(* IEC 61131-3 sources: AXOpen/src/components.rexroth.tightening/ctrl/src/TemplateComponent (part 2) *)

                    IF TRUE THEN
                        THIS.CallTimers(FALSE);
                        _progress := 346;
                    END_IF;
                END_IF;

                IF _progress = 346 THEN                                                                                     // TemplateTask_10steps_5 running: , <add the detailed description of the current action 7>
                    TaskMessenger.ActivateOnCondition(ULINT#546, _infoTimer.output, eAxoMessageCategory#Warning);
                    IF _infoTimer.output THEN
                        Status.Error.Id := UINT#546;
                    END_IF;

                    IF TRUE THEN
                        THIS.CallTimers(FALSE);
                        _progress := 347;
                    END_IF;
                END_IF;

                IF _progress = 347 THEN                                                                                     // TemplateTask_10steps_5 running: , <add the detailed description of the current action 8>
                    TaskMessenger.ActivateOnCondition(ULINT#547, _infoTimer.output, eAxoMessageCategory#Warning);
                    IF _infoTimer.output THEN
                        Status.Error.Id := UINT#547;
                    END_IF;

                    IF TRUE THEN
                        THIS.CallTimers(FALSE);
                        _progress := 348;
                    END_IF;
                END_IF;

                IF _progress = 348 THEN                                                                                     // TemplateTask_10steps_5 running: , <add the detailed description of the current action 9>
                    TaskMessenger.ActivateOnCondition(ULINT#548, _infoTimer.output, eAxoMessageCategory#Warning);
                    IF _infoTimer.output THEN
                        Status.Error.Id := UINT#548;
                    END_IF;

                    IF TRUE THEN
                        THIS.CallTimers(FALSE);
                        _progress := 349;
                    END_IF;
                END_IF;

                IF _progress = 349 THEN                                                                                     // TemplateTask_10steps_5 running: , <add the detailed description of the current action 10>
                    TemplateTask_10steps_5.DoneWhen(TRUE);
                END_IF;

                THIS.CallTimers(TRUE);

                TemplateTask_10steps_5.ThrowWhen(_errorTimer.output);
                Status.Action.Id := TO_UINT(_progress);
                TemplateTask_10steps_5.ThrowWhen(TemplateTask_10steps_5.Duration >= Config.ErrorTime ,'TemplateTask_10steps_5 error.');
            END_IF;
            IF TemplateTask_10steps_5.DoneReached() THEN
                Status.Action.Id :=  UINT#141;
                Status.Error.Id :=  UINT#0;
            ELSIF TemplateTask_10steps_5.ErrorOccured() THEN
                Status.Action.Id :=  UINT#940;
                Status.Error.Id  :=  UINT#940;
            ELSIF TemplateTask_10steps_5.AbortTriggered()THEN
                Status.Action.Id :=  UINT#941;
                Status.Error.Id  :=  UINT#941;
            END_IF;
            Messenger.ActivateOnCondition(ULINT#940,TemplateTask_10steps_5.HasError(), eAxoMessageCategory#Error);
            Messenger.ActivateOnCondition(ULINT#941,TemplateTask_10steps_5.IsAborted(), eAxoMessageCategory#Error);
            Messenger.ActivateOnCondition(ULINT#142,TemplateTask_10steps_5.RestoreTriggered() , eAxoMessageCategory#Error);
            IF TemplateTask_10steps_5.RestoreTriggered() AND _progress >= 340 AND _progress <= 349  THEN
                Status.Action.Id :=  UINT#142;
                _progress := 0;
            END_IF;
            //**************************************************

            //*************TemplateTask_10steps_6***************
            TemplateTask_10steps_6.SetIsDisabled(FALSE);
            IF TemplateTask_10steps_6.StartTriggered() THEN
                Status.Action.Id :=  UINT#150;
            END_IF;
            Messenger.ActivateOnCondition(ULINT#150,TemplateTask_10steps_6.IsBusy(), eAxoMessageCategory#Info);
            Messenger.ActivateOnCondition(ULINT#151,TemplateTask_10steps_6.IsDone(), eAxoMessageCategory#Info);
            IF TemplateTask_10steps_6.Execute(THIS) THEN
                IF _progress = 0 THEN
                    Status.Error.Id := UINT#0;
                    TaskMessenger.Restore();
                    THIS.CallTimers(FALSE);
                    _progress := 350;
                END_IF;

                IF _progress = 350 THEN                                                                                     // TemplateTask_10steps_6 running: , <add the detailed description of the current action 1>
                    TaskMessenger.ActivateOnCondition(ULINT#550, _infoTimer.output, eAxoMessageCategory#Warning);
                    IF _infoTimer.output THEN
                        Status.Error.Id := UINT#550;
                    END_IF;

                    IF TRUE THEN
                        THIS.CallTimers(FALSE);
                        _progress := 351;
                    END_IF;
                END_IF;

                IF _progress = 351 THEN                                                                                     // TemplateTask_10steps_6 running: , <add the detailed description of the current action 2>
                    TaskMessenger.ActivateOnCondition(ULINT#551, _infoTimer.output, eAxoMessageCategory#Warning);
                    IF _infoTimer.output THEN
                        Status.Error.Id := UINT#551;
                    END_IF;

                    IF TRUE THEN
                        THIS.CallTimers(FALSE);
                        _progress := 352;
                    END_IF;
                END_IF;

                IF _progress = 352 THEN                                                                                     // TemplateTask_10steps_6 running: , <add the detailed description of the current action 3>
                    TaskMessenger.ActivateOnCondition(ULINT#552, _infoTimer.output, eAxoMessageCategory#Warning);
                    IF _infoTimer.output THEN
                        Status.Error.Id := UINT#552;
                    END_IF;

                    IF TRUE THEN
                        THIS.CallTimers(FALSE);
                        _progress := 335;
                    END_IF;
                END_IF;

                IF _progress = 353 THEN                                                                                     // TemplateTask_10steps_6 running: , <add the detailed description of the current action 4>
                    TaskMessenger.ActivateOnCondition(ULINT#553, _infoTimer.output, eAxoMessageCategory#Warning);
                    IF _infoTimer.output THEN
                        Status.Error.Id := UINT#553;
                    END_IF;

                    IF TRUE THEN
                        THIS.CallTimers(FALSE);
                        _progress := 354;
                    END_IF;
                END_IF;

                IF _progress = 354 THEN                                                                                     // TemplateTask_10steps_6 running: , <add the detailed description of the current action 5>
                    TaskMessenger.ActivateOnCondition(ULINT#554, _infoTimer.output, eAxoMessageCategory#Warning);
                    IF _infoTimer.output THEN
                        Status.Error.Id := UINT#554;
                    END_IF;

                    IF TRUE THEN
                        THIS.CallTimers(FALSE);
                        _progress := 355;
                    END_IF;
                END_IF;

                IF _progress = 355 THEN                                                                                     // TemplateTask_10steps_6 running: , <add the detailed description of the current action 6>
                    TaskMessenger.ActivateOnCondition(ULINT#555, _infoTimer.output, eAxoMessageCategory#Warning);
                    IF _infoTimer.output THEN
                        Status.Error.Id := UINT#555;
                    END_IF;

                    IF TRUE THEN
                        THIS.CallTimers(FALSE);
                        _progress := 356;
                    END_IF;
                END_IF;

                IF _progress = 356 THEN                                                                                     // TemplateTask_10steps_6 running: , <add the detailed description of the current action 7>
                    TaskMessenger.ActivateOnCondition(ULINT#556, _infoTimer.output, eAxoMessageCategory#Warning);
                    IF _infoTimer.output THEN
                        Status.Error.Id := UINT#556;
                    END_IF;

                    IF TRUE THEN
                        THIS.CallTimers(FALSE);
                        _progress := 357;
                    END_IF;
                END_IF;

                IF _progress = 357 THEN                                                                                     // TemplateTask_10steps_6 running: , <add the detailed description of the current action 8>
                    TaskMessenger.ActivateOnCondition(ULINT#557, _infoTimer.output, eAxoMessageCategory#Warning);
                    IF _infoTimer.output THEN
                        Status.Error.Id := UINT#557;
                    END_IF;

                    IF TRUE THEN
                        THIS.CallTimers(FALSE);
                        _progress := 358;
                    END_IF;
                END_IF;

                IF _progress = 358 THEN                                                                                     // TemplateTask_10steps_6 running: , <add the detailed description of the current action 9>
                    TaskMessenger.ActivateOnCondition(ULINT#558, _infoTimer.output, eAxoMessageCategory#Warning);
                    IF _infoTimer.output THEN
                        Status.Error.Id := UINT#558;
                    END_IF;

                    IF TRUE THEN
                        THIS.CallTimers(FALSE);
                        _progress := 359;
                    END_IF;
                END_IF;

                IF _progress = 359 THEN                                                                                     // TemplateTask_10steps_6 running: , <add the detailed description of the current action 10>
                    TemplateTask_10steps_6.DoneWhen(TRUE);
                END_IF;

                THIS.CallTimers(TRUE);

                TemplateTask_10steps_6.ThrowWhen(_errorTimer.output);
                Status.Action.Id := TO_UINT(_progress);
                TemplateTask_10steps_6.ThrowWhen(TemplateTask_10steps_6.Duration >= Config.ErrorTime ,'TemplateTask_10steps_6 error.');
            END_IF;
            IF TemplateTask_10steps_6.DoneReached() THEN
                Status.Action.Id :=  UINT#151;
                Status.Error.Id :=  UINT#0;
            ELSIF TemplateTask_10steps_6.ErrorOccured() THEN
                Status.Action.Id :=  UINT#950;
                Status.Error.Id  :=  UINT#950;
            ELSIF TemplateTask_10steps_6.AbortTriggered()THEN
                Status.Action.Id :=  UINT#951;
                Status.Error.Id  :=  UINT#951;
            END_IF;
            Messenger.ActivateOnCondition(ULINT#950,TemplateTask_10steps_6.HasError(), eAxoMessageCategory#Error);
            Messenger.ActivateOnCondition(ULINT#951,TemplateTask_10steps_6.IsAborted(), eAxoMessageCategory#Error);
            Messenger.ActivateOnCondition(ULINT#152,TemplateTask_10steps_6.RestoreTriggered() , eAxoMessageCategory#Error);
            IF TemplateTask_10steps_6.RestoreTriggered() AND _progress >= 350 AND _progress <= 359  THEN
                Status.Action.Id :=  UINT#152;
                _progress := 0;
            END_IF;
            //**************************************************

            //*************TemplateTask_20steps_1***************
            TemplateTask_20steps_1.SetIsDisabled(FALSE);
            IF TemplateTask_20steps_1.StartTriggered() THEN
                Status.Action.Id :=  UINT#160;
            END_IF;
            Messenger.ActivateOnCondition(ULINT#160,TemplateTask_20steps_1.IsBusy(), eAxoMessageCategory#Info);
            Messenger.ActivateOnCondition(ULINT#161,TemplateTask_20steps_1.IsDone(), eAxoMessageCategory#Info);
            IF TemplateTask_20steps_1.Execute(THIS) THEN
                IF _progress = 0 THEN
                    Status.Error.Id := UINT#0;
                    TaskMessenger.Restore();
                    THIS.CallTimers(FALSE);
                    _progress := 360;
                END_IF;

                IF _progress = 360 THEN                                                                                     // TemplateTask_20steps_1 running: , <add the detailed description of the current action 1>
                    TaskMessenger.ActivateOnCondition(ULINT#560, _infoTimer.output, eAxoMessageCategory#Warning);
                    IF _infoTimer.output THEN
                        Status.Error.Id := UINT#560;
                    END_IF;

                    IF TRUE THEN
                        THIS.CallTimers(FALSE);
                        _progress := 361;
                    END_IF;
                END_IF;

                IF _progress = 361 THEN                                                                                     // TemplateTask_20steps_1 running: , <add the detailed description of the current action 2>
                    TaskMessenger.ActivateOnCondition(ULINT#561, _infoTimer.output, eAxoMessageCategory#Warning);
                    IF _infoTimer.output THEN
                        Status.Error.Id := UINT#561;
                    END_IF;

                    IF TRUE THEN
                        THIS.CallTimers(FALSE);
                        _progress := 362;
                    END_IF;
                END_IF;

                IF _progress = 362 THEN                                                                                     // TemplateTask_20steps_1 running: , <add the detailed description of the current action 3>
                    TaskMessenger.ActivateOnCondition(ULINT#562, _infoTimer.output, eAxoMessageCategory#Warning);
                    IF _infoTimer.output THEN
                        Status.Error.Id := UINT#562;
                    END_IF;

                    IF TRUE THEN
                        THIS.CallTimers(FALSE);
                        _progress := 363;
                    END_IF;
                END_IF;

                IF _progress = 363 THEN                                                                                     // TemplateTask_20steps_1 running: , <add the detailed description of the current action 4>
                    TaskMessenger.ActivateOnCondition(ULINT#563, _infoTimer.output, eAxoMessageCategory#Warning);
                    IF _infoTimer.output THEN
                        Status.Error.Id := UINT#563;
                    END_IF;

                    IF TRUE THEN
                        THIS.CallTimers(FALSE);
                        _progress := 364;
                    END_IF;
                END_IF;

                IF _progress = 364 THEN                                                                                     // TemplateTask_20steps_1 running: , <add the detailed description of the current action 5>
                    TaskMessenger.ActivateOnCondition(ULINT#564, _infoTimer.output, eAxoMessageCategory#Warning);
                    IF _infoTimer.output THEN
                        Status.Error.Id := UINT#564;
                    END_IF;

                    IF TRUE THEN
                        THIS.CallTimers(FALSE);
                        _progress := 365;
                    END_IF;
                END_IF;

                IF _progress = 365 THEN                                                                                     // TemplateTask_20steps_1 running: , <add the detailed description of the current action 6>
                    TaskMessenger.ActivateOnCondition(ULINT#565, _infoTimer.output, eAxoMessageCategory#Warning);
                    IF _infoTimer.output THEN
                        Status.Error.Id := UINT#565;
                    END_IF;

                    IF TRUE THEN
                        THIS.CallTimers(FALSE);
                        _progress := 366;
                    END_IF;
                END_IF;

                IF _progress = 366 THEN                                                                                     // TemplateTask_20steps_1 running: , <add the detailed description of the current action 7>
                    TaskMessenger.ActivateOnCondition(ULINT#566, _infoTimer.output, eAxoMessageCategory#Warning);
                    IF _infoTimer.output THEN
                        Status.Error.Id := UINT#566;
                    END_IF;

                    IF TRUE THEN
                        THIS.CallTimers(FALSE);
                        _progress := 367;
                    END_IF;
                END_IF;

                IF _progress = 367 THEN                                                                                     // TemplateTask_20steps_1 running: , <add the detailed description of the current action 8>
                    TaskMessenger.ActivateOnCondition(ULINT#567, _infoTimer.output, eAxoMessageCategory#Warning);
                    IF _infoTimer.output THEN
                        Status.Error.Id := UINT#567;
                    END_IF;

                    IF TRUE THEN
                        THIS.CallTimers(FALSE);
                        _progress := 368;
                    END_IF;
                END_IF;

                IF _progress = 368 THEN                                                                                     // TemplateTask_20steps_1 running: , <add the detailed description of the current action 9>
                    TaskMessenger.ActivateOnCondition(ULINT#568, _infoTimer.output, eAxoMessageCategory#Warning);
                    IF _infoTimer.output THEN
                        Status.Error.Id := UINT#568;
                    END_IF;

                    IF TRUE THEN
                        THIS.CallTimers(FALSE);
                        _progress := 369;
                    END_IF;
                END_IF;

                IF _progress = 369 THEN                                                                                     // TemplateTask_20steps_1 running: , <add the detailed description of the current action 10>
                    TaskMessenger.ActivateOnCondition(ULINT#569, _infoTimer.output, eAxoMessageCategory#Warning);
                    IF _infoTimer.output THEN
                        Status.Error.Id := UINT#569;
                    END_IF;

                    IF TRUE THEN
                        THIS.CallTimers(FALSE);
                        _progress := 370;
                    END_IF;
                END_IF;

                IF _progress = 370 THEN                                                                                     // TemplateTask_20steps_1 running: , <add the detailed description of the current action 11>
                    TaskMessenger.ActivateOnCondition(ULINT#570, _infoTimer.output, eAxoMessageCategory#Warning);
                    IF _infoTimer.output THEN
                        Status.Error.Id := UINT#570;
                    END_IF;

                    IF TRUE THEN
                        THIS.CallTimers(FALSE);
                        _progress := 371;
                    END_IF;
                END_IF;

                IF _progress = 371 THEN                                                                                     // TemplateTask_20steps_1 running: , <add the detailed description of the current action 12>
                    TaskMessenger.ActivateOnCondition(ULINT#571, _infoTimer.output, eAxoMessageCategory#Warning);
                    IF _infoTimer.output THEN
                        Status.Error.Id := UINT#571;
                    END_IF;

                    IF TRUE THEN
                        THIS.CallTimers(FALSE);
                        _progress := 372;
                    END_IF;
                END_IF;

                IF _progress = 372 THEN                                                                                     // TemplateTask_20steps_1 running: , <add the detailed description of the current action 13>
                    TaskMessenger.ActivateOnCondition(ULINT#572, _infoTimer.output, eAxoMessageCategory#Warning);
                    IF _infoTimer.output THEN
                        Status.Error.Id := UINT#572;
                    END_IF;

                    IF TRUE THEN
                        THIS.CallTimers(FALSE);
                        _progress := 373;
                    END_IF;
                END_IF;

                IF _progress = 373 THEN                                                                                     // TemplateTask_20steps_1 running: , <add the detailed description of the current action 14>
                    TaskMessenger.ActivateOnCondition(ULINT#573, _infoTimer.output, eAxoMessageCategory#Warning);
                    IF _infoTimer.output THEN
                        Status.Error.Id := UINT#573;
                    END_IF;

                    IF TRUE THEN
                        THIS.CallTimers(FALSE);
                        _progress := 374;
                    END_IF;
                END_IF;

                IF _progress = 374 THEN                                                                                     // TemplateTask_20steps_1 running: , <add the detailed description of the current action 15>
                    TaskMessenger.ActivateOnCondition(ULINT#574, _infoTimer.output, eAxoMessageCategory#Warning);
                    IF _infoTimer.output THEN
                        Status.Error.Id := UINT#574;
                    END_IF;

                    IF TRUE THEN
                        THIS.CallTimers(FALSE);
                        _progress := 375;
                    END_IF;
                END_IF;

                IF _progress = 375 THEN                                                                                     // TemplateTask_20steps_1 running: , <add the detailed description of the current action 16>
                    TaskMessenger.ActivateOnCondition(ULINT#575, _infoTimer.output, eAxoMessageCategory#Warning);
                    IF _infoTimer.output THEN
                        Status.Error.Id := UINT#575;
                    END_IF;

                    IF TRUE THEN
                        THIS.CallTimers(FALSE);
                        _progress := 376;
                    END_IF;
                END_IF;

                IF _progress = 376 THEN                                                                                     // TemplateTask_20steps_1 running: , <add the detailed description of the current action 17>
                    TaskMessenger.ActivateOnCondition(ULINT#576, _infoTimer.output, eAxoMessageCategory#Warning);
                    IF _infoTimer.output THEN
                        Status.Error.Id := UINT#576;
                    END_IF;

                    IF TRUE THEN
                        THIS.CallTimers(FALSE);
                        _progress := 377;
                    END_IF;
                END_IF;

                IF _progress = 377 THEN                                                                                     // TemplateTask_20steps_1 running: , <add the detailed description of the current action 18>
                    TaskMessenger.ActivateOnCondition(ULINT#577, _infoTimer.output, eAxoMessageCategory#Warning);
                    IF _infoTimer.output THEN
                        Status.Error.Id := UINT#577;
                    END_IF;

                    IF TRUE THEN
                        THIS.CallTimers(FALSE);
                        _progress := 378;
                    END_IF;
                END_IF;

                IF _progress = 378 THEN                                                                                     // TemplateTask_20steps_1 running: , <add the detailed description of the current action 19>
                    TaskMessenger.ActivateOnCondition(ULINT#578, _infoTimer.output, eAxoMessageCategory#Warning);
                    IF _infoTimer.output THEN
                        Status.Error.Id := UINT#578;
                    END_IF;

                    IF TRUE THEN
                        THIS.CallTimers(FALSE);
                        _progress := 379;
                    END_IF;
                END_IF;

                IF _progress = 379 THEN                                                                                     // TemplateTask_20steps_1 running: , <add the detailed description of the current action 20>
                    TemplateTask_20steps_1.DoneWhen(TRUE);
                END_IF;

                THIS.CallTimers(TRUE);

                TemplateTask_20steps_1.ThrowWhen(_errorTimer.output);
                Status.Action.Id := TO_UINT(_progress);
                TemplateTask_20steps_1.ThrowWhen(TemplateTask_20steps_1.Duration >= Config.ErrorTime ,'TemplateTask_20steps_1 error.');
            END_IF;
            IF TemplateTask_20steps_1.DoneReached() THEN
                Status.Action.Id :=  UINT#161;
                Status.Error.Id :=  UINT#0;
            ELSIF TemplateTask_20steps_1.ErrorOccured() THEN
                Status.Action.Id :=  UINT#960;
                Status.Error.Id  :=  UINT#960;
            ELSIF TemplateTask_20steps_1.AbortTriggered()THEN
                Status.Action.Id :=  UINT#961;
                Status.Error.Id  :=  UINT#961;
            END_IF;
            Messenger.ActivateOnCondition(ULINT#960,TemplateTask_20steps_1.HasError(), eAxoMessageCategory#Error);
            Messenger.ActivateOnCondition(ULINT#961,TemplateTask_20steps_1.IsAborted(), eAxoMessageCategory#Error);
            Messenger.ActivateOnCondition(ULINT#162,TemplateTask_20steps_1.RestoreTriggered() , eAxoMessageCategory#Error);
            IF TemplateTask_20steps_1.RestoreTriggered() AND _progress >= 360 AND _progress <= 379  THEN
                Status.Action.Id :=  UINT#162;
                _progress := 0;
            END_IF;
            //**************************************************

            //*************TemplateTask_20steps_2***************
            TemplateTask_20steps_2.SetIsDisabled(FALSE);
            IF TemplateTask_20steps_2.StartTriggered() THEN
                Status.Action.Id :=  UINT#180;
            END_IF;
            Messenger.ActivateOnCondition(ULINT#180,TemplateTask_20steps_2.IsBusy(), eAxoMessageCategory#Info);
            Messenger.ActivateOnCondition(ULINT#181,TemplateTask_20steps_2.IsDone(), eAxoMessageCategory#Info);
            IF TemplateTask_20steps_2.Execute(THIS) THEN
                IF _progress = 0 THEN
                    Status.Error.Id := UINT#0;
                    TaskMessenger.Restore();
                    THIS.CallTimers(FALSE);
                    _progress := 380;
                END_IF;

                IF _progress = 380 THEN                                                                                     // TemplateTask_20steps_2 running: , <add the detailed description of the current action 1>
                    TaskMessenger.ActivateOnCondition(ULINT#580, _infoTimer.output, eAxoMessageCategory#Warning);
                    IF _infoTimer.output THEN
                        Status.Error.Id := UINT#580;
                    END_IF;

                    IF TRUE THEN
                        THIS.CallTimers(FALSE);
                        _progress := 381;
                    END_IF;
                END_IF;

                IF _progress = 381 THEN                                                                                     // TemplateTask_20steps_2 running: , <add the detailed description of the current action 2>
                    TaskMessenger.ActivateOnCondition(ULINT#581, _infoTimer.output, eAxoMessageCategory#Warning);
                    IF _infoTimer.output THEN
                        Status.Error.Id := UINT#581;
                    END_IF;

                    IF TRUE THEN
                        THIS.CallTimers(FALSE);
                        _progress := 382;
                    END_IF;
                END_IF;

                IF _progress = 382 THEN                                                                                     // TemplateTask_20steps_2 running: , <add the detailed description of the current action 3>
                    TaskMessenger.ActivateOnCondition(ULINT#582, _infoTimer.output, eAxoMessageCategory#Warning);
                    IF _infoTimer.output THEN
                        Status.Error.Id := UINT#582;
                    END_IF;

                    IF TRUE THEN
                        THIS.CallTimers(FALSE);
                        _progress := 383;
                    END_IF;
                END_IF;

                IF _progress = 383 THEN                                                                                     // TemplateTask_20steps_2 running: , <add the detailed description of the current action 4>
                    TaskMessenger.ActivateOnCondition(ULINT#583, _infoTimer.output, eAxoMessageCategory#Warning);
                    IF _infoTimer.output THEN
                        Status.Error.Id := UINT#583;
                    END_IF;

                    IF TRUE THEN
                        THIS.CallTimers(FALSE);
                        _progress := 384;
                    END_IF;
                END_IF;

                IF _progress = 384 THEN                                                                                     // TemplateTask_20steps_2 running: , <add the detailed description of the current action 5>
                    TaskMessenger.ActivateOnCondition(ULINT#584, _infoTimer.output, eAxoMessageCategory#Warning);
                    IF _infoTimer.output THEN
                        Status.Error.Id := UINT#584;
                    END_IF;

                    IF TRUE THEN
                        THIS.CallTimers(FALSE);
                        _progress := 385;
                    END_IF;
                END_IF;

                IF _progress = 385 THEN                                                                                     // TemplateTask_20steps_2 running: , <add the detailed description of the current action 6>
                    TaskMessenger.ActivateOnCondition(ULINT#585, _infoTimer.output, eAxoMessageCategory#Warning);
                    IF _infoTimer.output THEN
                        Status.Error.Id := UINT#585;
                    END_IF;

                    IF TRUE THEN
                        THIS.CallTimers(FALSE);
                        _progress := 386;
                    END_IF;
                END_IF;

                IF _progress = 386 THEN                                                                                     // TemplateTask_20steps_2 running: , <add the detailed description of the current action 7>
                    TaskMessenger.ActivateOnCondition(ULINT#586, _infoTimer.output, eAxoMessageCategory#Warning);
                    IF _infoTimer.output THEN
                        Status.Error.Id := UINT#586;
                    END_IF;

                    IF TRUE THEN
                        THIS.CallTimers(FALSE);
                        _progress := 387;
                    END_IF;
                END_IF;

                IF _progress = 387 THEN                                                                                     // TemplateTask_20steps_2 running: , <add the detailed description of the current action 8>
                    TaskMessenger.ActivateOnCondition(ULINT#587, _infoTimer.output, eAxoMessageCategory#Warning);
                    IF _infoTimer.output THEN
                        Status.Error.Id := UINT#587;
                    END_IF;

                    IF TRUE THEN
                        THIS.CallTimers(FALSE);
                        _progress := 388;
                    END_IF;
                END_IF;

                IF _progress = 388 THEN                                                                                     // TemplateTask_20steps_2 running: , <add the detailed description of the current action 9>
                    TaskMessenger.ActivateOnCondition(ULINT#588, _infoTimer.output, eAxoMessageCategory#Warning);
                    IF _infoTimer.output THEN
                        Status.Error.Id := UINT#588;
                    END_IF;

                    IF TRUE THEN
                        THIS.CallTimers(FALSE);
                        _progress := 389;
                    END_IF;
                END_IF;

                IF _progress = 389 THEN                                                                                     // TemplateTask_20steps_2 running: , <add the detailed description of the current action 10>
                    TaskMessenger.ActivateOnCondition(ULINT#589, _infoTimer.output, eAxoMessageCategory#Warning);
                    IF _infoTimer.output THEN
                        Status.Error.Id := UINT#589;
                    END_IF;

                    IF TRUE THEN
                        THIS.CallTimers(FALSE);
                        _progress := 390;
                    END_IF;
                END_IF;

                IF _progress = 390 THEN                                                                                     // TemplateTask_20steps_2 running: , <add the detailed description of the current action 11>
                    TaskMessenger.ActivateOnCondition(ULINT#590, _infoTimer.output, eAxoMessageCategory#Warning);
                    IF _infoTimer.output THEN
                        Status.Error.Id := UINT#590;
                    END_IF;

                    IF TRUE THEN
                        THIS.CallTimers(FALSE);
                        _progress := 391;
                    END_IF;
                END_IF;

                IF _progress = 391 THEN                                                                                     // TemplateTask_20steps_2 running: , <add the detailed description of the current action 12>
                    TaskMessenger.ActivateOnCondition(ULINT#591, _infoTimer.output, eAxoMessageCategory#Warning);
                    IF _infoTimer.output THEN
                        Status.Error.Id := UINT#591;
                    END_IF;

                    IF TRUE THEN
                        THIS.CallTimers(FALSE);
                        _progress := 392;
                    END_IF;
                END_IF;

                IF _progress = 392 THEN                                                                                     // TemplateTask_20steps_2 running: , <add the detailed description of the current action 13>
                    TaskMessenger.ActivateOnCondition(ULINT#592, _infoTimer.output, eAxoMessageCategory#Warning);
                    IF _infoTimer.output THEN
                        Status.Error.Id := UINT#592;
                    END_IF;

                    IF TRUE THEN
                        THIS.CallTimers(FALSE);
                        _progress := 393;
                    END_IF;
                END_IF;

                IF _progress = 393 THEN                                                                                     // TemplateTask_20steps_2 running: , <add the detailed description of the current action 14>
                    TaskMessenger.ActivateOnCondition(ULINT#593, _infoTimer.output, eAxoMessageCategory#Warning);
                    IF _infoTimer.output THEN
                        Status.Error.Id := UINT#593;
                    END_IF;

                    IF TRUE THEN
                        THIS.CallTimers(FALSE);
                        _progress := 394;
                    END_IF;
                END_IF;

                IF _progress = 394 THEN                                                                                     // TemplateTask_20steps_2 running: , <add the detailed description of the current action 15>
                    TaskMessenger.ActivateOnCondition(ULINT#594, _infoTimer.output, eAxoMessageCategory#Warning);
                    IF _infoTimer.output THEN
                        Status.Error.Id := UINT#594;
                    END_IF;

                    IF TRUE THEN
                        THIS.CallTimers(FALSE);
                        _progress := 395;
                    END_IF;
                END_IF;

                IF _progress = 395 THEN                                                                                     // TemplateTask_20steps_2 running: , <add the detailed description of the current action 16>
                    TaskMessenger.ActivateOnCondition(ULINT#595, _infoTimer.output, eAxoMessageCategory#Warning);
                    IF _infoTimer.output THEN
                        Status.Error.Id := UINT#595;
                    END_IF;

                    IF TRUE THEN
                        THIS.CallTimers(FALSE);
                        _progress := 396;
                    END_IF;
                END_IF;

                IF _progress = 396 THEN                                                                                     // TemplateTask_20steps_2 running: , <add the detailed description of the current action 17>
                    TaskMessenger.ActivateOnCondition(ULINT#596, _infoTimer.output, eAxoMessageCategory#Warning);
                    IF _infoTimer.output THEN
                        Status.Error.Id := UINT#596;
                    END_IF;

                    IF TRUE THEN
                        THIS.CallTimers(FALSE);
                        _progress := 397;
                    END_IF;
                END_IF;

                IF _progress = 397 THEN                                                                                     // TemplateTask_20steps_2 running: , <add the detailed description of the current action 18>
                    TaskMessenger.ActivateOnCondition(ULINT#597, _infoTimer.output, eAxoMessageCategory#Warning);
                    IF _infoTimer.output THEN
                        Status.Error.Id := UINT#597;
                    END_IF;

                    IF TRUE THEN
                        THIS.CallTimers(FALSE);
                        _progress := 398;
                    END_IF;
                END_IF;

                IF _progress = 398 THEN                                                                                     // TemplateTask_20steps_2 running: , <add the detailed description of the current action 19>
                    TaskMessenger.ActivateOnCondition(ULINT#598, _infoTimer.output, eAxoMessageCategory#Warning);
                    IF _infoTimer.output THEN
                        Status.Error.Id := UINT#598;
                    END_IF;

                    IF TRUE THEN
                        THIS.CallTimers(FALSE);
                        _progress := 399;
                    END_IF;
                END_IF;

                IF _progress = 399 THEN                                                                                     // TemplateTask_20steps_2 running: , <add the detailed description of the current action 20>
                    TemplateTask_20steps_2.DoneWhen(TRUE);
                END_IF;

                THIS.CallTimers(TRUE);

                TemplateTask_20steps_2.ThrowWhen(_errorTimer.output);
                Status.Action.Id := TO_UINT(_progress);
                TemplateTask_20steps_2.ThrowWhen(TemplateTask_20steps_2.Duration >= Config.ErrorTime ,'TemplateTask_20steps_2 error.');
            END_IF;
            IF TemplateTask_20steps_2.DoneReached() THEN
                Status.Action.Id :=  UINT#181;
                Status.Error.Id :=  UINT#0;
            ELSIF TemplateTask_20steps_2.ErrorOccured() THEN
                Status.Action.Id :=  UINT#980;
                Status.Error.Id  :=  UINT#980;
            ELSIF TemplateTask_20steps_2.AbortTriggered()THEN
                Status.Action.Id :=  UINT#981;
                Status.Error.Id  :=  UINT#981;
            END_IF;
            Messenger.ActivateOnCondition(ULINT#980,TemplateTask_20steps_2.HasError(), eAxoMessageCategory#Error);
            Messenger.ActivateOnCondition(ULINT#981,TemplateTask_20steps_2.IsAborted(), eAxoMessageCategory#Error);
            Messenger.ActivateOnCondition(ULINT#182,TemplateTask_20steps_2.RestoreTriggered() , eAxoMessageCategory#Error);
            IF TemplateTask_20steps_2.RestoreTriggered() AND _progress >= 380 AND _progress <= 399  THEN
                Status.Action.Id :=  UINT#182;
                _progress := 0;
            END_IF;
            //**************************************************

            //*************TemplateTask_20steps_3***************
            TemplateTask_20steps_3.SetIsDisabled(FALSE);
            IF TemplateTask_20steps_3.StartTriggered() THEN
                Status.Action.Id :=  UINT#200;
            END_IF;
            Messenger.ActivateOnCondition(ULINT#200,TemplateTask_20steps_3.IsBusy(), eAxoMessageCategory#Info);
            Messenger.ActivateOnCondition(ULINT#201,TemplateTask_20steps_3.IsDone(), eAxoMessageCategory#Info);
            IF TemplateTask_20steps_3.Execute(THIS) THEN
                IF _progress = 0 THEN
                    Status.Error.Id := UINT#0;
                    TaskMessenger.Restore();
                    THIS.CallTimers(FALSE);
                    _progress := 400;
                END_IF;

                IF _progress = 400 THEN                                                                                     // TemplateTask_20steps_3 running: , <add the detailed description of the current action 1>
                    TaskMessenger.ActivateOnCondition(ULINT#600, _infoTimer.output, eAxoMessageCategory#Warning);
                    IF _infoTimer.output THEN
                        Status.Error.Id := UINT#600;
                    END_IF;

                    IF TRUE THEN
                        THIS.CallTimers(FALSE);
                        _progress := 401;
                    END_IF;
                END_IF;

                IF _progress = 401 THEN                                                                                     // TemplateTask_20steps_3 running: , <add the detailed description of the current action 2>
                    TaskMessenger.ActivateOnCondition(ULINT#601, _infoTimer.output, eAxoMessageCategory#Warning);
                    IF _infoTimer.output THEN
                        Status.Error.Id := UINT#601;
                    END_IF;

                    IF TRUE THEN
                        THIS.CallTimers(FALSE);
                        _progress := 402;
                    END_IF;
                END_IF;

                IF _progress = 402 THEN                                                                                     // TemplateTask_20steps_3 running: , <add the detailed description of the current action 3>
                    TaskMessenger.ActivateOnCondition(ULINT#602, _infoTimer.output, eAxoMessageCategory#Warning);
                    IF _infoTimer.output THEN
                        Status.Error.Id := UINT#602;
                    END_IF;

                    IF TRUE THEN
                        THIS.CallTimers(FALSE);
                        _progress := 403;
                    END_IF;
                END_IF;

                IF _progress = 403 THEN                                                                                     // TemplateTask_20steps_3 running: , <add the detailed description of the current action 4>
                    TaskMessenger.ActivateOnCondition(ULINT#603, _infoTimer.output, eAxoMessageCategory#Warning);
                    IF _infoTimer.output THEN
                        Status.Error.Id := UINT#603;
                    END_IF;

                    IF TRUE THEN
                        THIS.CallTimers(FALSE);
                        _progress := 404;
                    END_IF;
                END_IF;

                IF _progress = 404 THEN                                                                                     // TemplateTask_20steps_3 running: , <add the detailed description of the current action 5>
                    TaskMessenger.ActivateOnCondition(ULINT#604, _infoTimer.output, eAxoMessageCategory#Warning);
                    IF _infoTimer.output THEN
                        Status.Error.Id := UINT#604;
                    END_IF;

                    IF TRUE THEN
                        THIS.CallTimers(FALSE);
                        _progress := 405;
                    END_IF;
                END_IF;

                IF _progress = 405 THEN                                                                                     // TemplateTask_20steps_3 running: , <add the detailed description of the current action 6>
                    TaskMessenger.ActivateOnCondition(ULINT#605, _infoTimer.output, eAxoMessageCategory#Warning);
                    IF _infoTimer.output THEN
                        Status.Error.Id := UINT#605;
                    END_IF;

                    IF TRUE THEN
                        THIS.CallTimers(FALSE);
                        _progress := 406;
                    END_IF;
                END_IF;

                IF _progress = 406 THEN                                                                                     // TemplateTask_20steps_3 running: , <add the detailed description of the current action 7>
                    TaskMessenger.ActivateOnCondition(ULINT#606, _infoTimer.output, eAxoMessageCategory#Warning);
                    IF _infoTimer.output THEN
                        Status.Error.Id := UINT#606;
                    END_IF;

                    IF TRUE THEN
                        THIS.CallTimers(FALSE);
                        _progress := 407;
                    END_IF;
                END_IF;

                IF _progress = 407 THEN                                                                                     // TemplateTask_20steps_3 running: , <add the detailed description of the current action 8>
                    TaskMessenger.ActivateOnCondition(ULINT#607, _infoTimer.output, eAxoMessageCategory#Warning);
                    IF _infoTimer.output THEN
                        Status.Error.Id := UINT#607;
                    END_IF;

                    IF TRUE THEN
                        THIS.CallTimers(FALSE);
                        _progress := 408;
                    END_IF;
                END_IF;

                IF _progress = 408 THEN                                                                                     // TemplateTask_20steps_3 running: , <add the detailed description of the current action 9>
                    TaskMessenger.ActivateOnCondition(ULINT#608, _infoTimer.output, eAxoMessageCategory#Warning);
                    IF _infoTimer.output THEN
                        Status.Error.Id := UINT#608;
                    END_IF;

                    IF TRUE THEN
                        THIS.CallTimers(FALSE);
                        _progress := 409;
                    END_IF;
                END_IF;

                IF _progress = 409 THEN                                                                                     // TemplateTask_20steps_3 running: , <add the detailed description of the current action 10>
                    TaskMessenger.ActivateOnCondition(ULINT#609, _infoTimer.output, eAxoMessageCategory#Warning);
                    IF _infoTimer.output THEN
                        Status.Error.Id := UINT#609;
                    END_IF;

                    IF TRUE THEN
                        THIS.CallTimers(FALSE);
                        _progress := 410;
                    END_IF;
                END_IF;

                IF _progress = 410 THEN                                                                                     // TemplateTask_20steps_3 running: , <add the detailed description of the current action 11>
                    TaskMessenger.ActivateOnCondition(ULINT#610, _infoTimer.output, eAxoMessageCategory#Warning);
                    IF _infoTimer.output THEN
                        Status.Error.Id := UINT#610;
                    END_IF;

                    IF TRUE THEN
                        THIS.CallTimers(FALSE);
                        _progress := 411;
                    END_IF;
                END_IF;

                IF _progress = 411 THEN                                                                                     // TemplateTask_20steps_3 running: , <add the detailed description of the current action 12>
                    TaskMessenger.ActivateOnCondition(ULINT#611, _infoTimer.output, eAxoMessageCategory#Warning);
                    IF _infoTimer.output THEN
                        Status.Error.Id := UINT#611;
                    END_IF;

                    IF TRUE THEN
                        THIS.CallTimers(FALSE);
                        _progress := 412;
                    END_IF;
                END_IF;

                IF _progress = 412 THEN                                                                                     // TemplateTask_20steps_3 running: , <add the detailed description of the current action 13>
                    TaskMessenger.ActivateOnCondition(ULINT#612, _infoTimer.output, eAxoMessageCategory#Warning);
                    IF _infoTimer.output THEN
                        Status.Error.Id := UINT#612;
                    END_IF;

                    IF TRUE THEN
                        THIS.CallTimers(FALSE);
                        _progress := 413;
                    END_IF;
                END_IF;

                IF _progress = 413 THEN                                                                                     // TemplateTask_20steps_3 running: , <add the detailed description of the current action 14>
                    TaskMessenger.ActivateOnCondition(ULINT#613, _infoTimer.output, eAxoMessageCategory#Warning);
                    IF _infoTimer.output THEN
                        Status.Error.Id := UINT#613;
                    END_IF;

                    IF TRUE THEN
                        THIS.CallTimers(FALSE);
                        _progress := 414;
                    END_IF;
                END_IF;

                IF _progress = 414 THEN                                                                                     // TemplateTask_20steps_3 running: , <add the detailed description of the current action 15>
                    TaskMessenger.ActivateOnCondition(ULINT#614, _infoTimer.output, eAxoMessageCategory#Warning);
                    IF _infoTimer.output THEN
                        Status.Error.Id := UINT#614;
                    END_IF;

                    IF TRUE THEN
                        THIS.CallTimers(FALSE);
                        _progress := 415;
                    END_IF;
                END_IF;

                IF _progress = 415 THEN                                                                                     // TemplateTask_20steps_3 running: , <add the detailed description of the current action 16>
                    TaskMessenger.ActivateOnCondition(ULINT#615, _infoTimer.output, eAxoMessageCategory#Warning);
                    IF _infoTimer.output THEN
                        Status.Error.Id := UINT#615;
                    END_IF;

                    IF TRUE THEN
                        THIS.CallTimers(FALSE);
                        _progress := 416;
                    END_IF;
                END_IF;

                IF _progress = 416 THEN                                                                                     // TemplateTask_20steps_3 running: , <add the detailed description of the current action 17>
                    TaskMessenger.ActivateOnCondition(ULINT#616, _infoTimer.output, eAxoMessageCategory#Warning);
                    IF _infoTimer.output THEN
                        Status.Error.Id := UINT#616;
                    END_IF;

                    IF TRUE THEN
                        THIS.CallTimers(FALSE);
                        _progress := 417;
                    END_IF;
                END_IF;

                IF _progress = 417 THEN                                                                                     // TemplateTask_20steps_3 running: , <add the detailed description of the current action 18>
                    TaskMessenger.ActivateOnCondition(ULINT#617, _infoTimer.output, eAxoMessageCategory#Warning);
                    IF _infoTimer.output THEN
                        Status.Error.Id := UINT#617;
                    END_IF;

                    IF TRUE THEN
                        THIS.CallTimers(FALSE);
                        _progress := 418;
                    END_IF;
                END_IF;

                IF _progress = 418 THEN                                                                                     // TemplateTask_20steps_3 running: , <add the detailed description of the current action 19>
                    TaskMessenger.ActivateOnCondition(ULINT#618, _infoTimer.output, eAxoMessageCategory#Warning);
                    IF _infoTimer.output THEN
                        Status.Error.Id := UINT#618;
                    END_IF;

                    IF TRUE THEN
                        THIS.CallTimers(FALSE);
                        _progress := 419;
                    END_IF;
                END_IF;

                IF _progress = 419 THEN                                                                                     // TemplateTask_20steps_3 running: , <add the detailed description of the current action 20>
                    TemplateTask_20steps_3.DoneWhen(TRUE);
                END_IF;

                THIS.CallTimers(TRUE);

                TemplateTask_20steps_3.ThrowWhen(_errorTimer.output);
                Status.Action.Id := TO_UINT(_progress);
                TemplateTask_20steps_3.ThrowWhen(TemplateTask_20steps_3.Duration >= Config.ErrorTime ,'TemplateTask_20steps_3 error.');
            END_IF;
            IF TemplateTask_20steps_3.DoneReached() THEN
                Status.Action.Id :=  UINT#201;
                Status.Error.Id :=  UINT#0;
            ELSIF TemplateTask_20steps_3.ErrorOccured() THEN
                Status.Action.Id :=  UINT#1000;
                Status.Error.Id  :=  UINT#1000;
            ELSIF TemplateTask_20steps_3.AbortTriggered()THEN
                Status.Action.Id :=  UINT#1001;
                Status.Error.Id  :=  UINT#1001;
            END_IF;
            Messenger.ActivateOnCondition(ULINT#1000,TemplateTask_20steps_3.HasError(), eAxoMessageCategory#Error);
            Messenger.ActivateOnCondition(ULINT#1001,TemplateTask_20steps_3.IsAborted(), eAxoMessageCategory#Error);
            Messenger.ActivateOnCondition(ULINT#202,TemplateTask_20steps_3.RestoreTriggered() , eAxoMessageCategory#Error);
            IF TemplateTask_20steps_3.RestoreTriggered() AND _progress >= 400 AND _progress <= 419  THEN
                Status.Action.Id :=  UINT#202;
                _progress := 0;
            END_IF;
            //**************************************************

            //*************TemplateTask_20steps_4***************
            TemplateTask_20steps_4.SetIsDisabled(FALSE);
            IF TemplateTask_20steps_4.StartTriggered() THEN
                Status.Action.Id :=  UINT#220;
            END_IF;
            Messenger.ActivateOnCondition(ULINT#220,TemplateTask_20steps_4.IsBusy(), eAxoMessageCategory#Info);
            Messenger.ActivateOnCondition(ULINT#221,TemplateTask_20steps_4.IsDone(), eAxoMessageCategory#Info);
            IF TemplateTask_20steps_4.Execute(THIS) THEN
                IF _progress = 0 THEN
                    Status.Error.Id := UINT#0;
                    TaskMessenger.Restore();
                    THIS.CallTimers(FALSE);
                    _progress := 420;
                END_IF;

                IF _progress = 420 THEN                                                                                     // TemplateTask_20steps_4 running: , <add the detailed description of the current action 1>
                    TaskMessenger.ActivateOnCondition(ULINT#620, _infoTimer.output, eAxoMessageCategory#Warning);
                    IF _infoTimer.output THEN
                        Status.Error.Id := UINT#620;
                    END_IF;

                    IF TRUE THEN
                        THIS.CallTimers(FALSE);
                        _progress := 421;
                    END_IF;
                END_IF;

                IF _progress = 421 THEN                                                                                     // TemplateTask_20steps_4 running: , <add the detailed description of the current action 2>
                    TaskMessenger.ActivateOnCondition(ULINT#621, _infoTimer.output, eAxoMessageCategory#Warning);
                    IF _infoTimer.output THEN
                        Status.Error.Id := UINT#621;
                    END_IF;

                    IF TRUE THEN
                        THIS.CallTimers(FALSE);
                        _progress := 422;
                    END_IF;
                END_IF;

                IF _progress = 422 THEN                                                                                     // TemplateTask_20steps_4 running: , <add the detailed description of the current action 3>
                    TaskMessenger.ActivateOnCondition(ULINT#622, _infoTimer.output, eAxoMessageCategory#Warning);
                    IF _infoTimer.output THEN
                        Status.Error.Id := UINT#622;
                    END_IF;

                    IF TRUE THEN
                        THIS.CallTimers(FALSE);
                        _progress := 423;
                    END_IF;
                END_IF;

                IF _progress = 423 THEN                                                                                     // TemplateTask_20steps_4 running: , <add the detailed description of the current action 4>
                    TaskMessenger.ActivateOnCondition(ULINT#623, _infoTimer.output, eAxoMessageCategory#Warning);
                    IF _infoTimer.output THEN
                        Status.Error.Id := UINT#623;
                    END_IF;

                    IF TRUE THEN
                        THIS.CallTimers(FALSE);
                        _progress := 424;
                    END_IF;
                END_IF;

                IF _progress = 424 THEN                                                                                     // TemplateTask_20steps_4 running: , <add the detailed description of the current action 5>
                    TaskMessenger.ActivateOnCondition(ULINT#624, _infoTimer.output, eAxoMessageCategory#Warning);
                    IF _infoTimer.output THEN
                        Status.Error.Id := UINT#624;
                    END_IF;

                    IF TRUE THEN
                        THIS.CallTimers(FALSE);
                        _progress := 425;
                    END_IF;
                END_IF;

                IF _progress = 425 THEN                                                                                     // TemplateTask_20steps_4 running: , <add the detailed description of the current action 6>
                    TaskMessenger.ActivateOnCondition(ULINT#625, _infoTimer.output, eAxoMessageCategory#Warning);
                    IF _infoTimer.output THEN
                        Status.Error.Id := UINT#625;
                    END_IF;

                    IF TRUE THEN
                        THIS.CallTimers(FALSE);
                        _progress := 426;
                    END_IF;
                END_IF;

                IF _progress = 426 THEN                                                                                     // TemplateTask_20steps_4 running: , <add the detailed description of the current action 7>
                    TaskMessenger.ActivateOnCondition(ULINT#626, _infoTimer.output, eAxoMessageCategory#Warning);
                    IF _infoTimer.output THEN
                        Status.Error.Id := UINT#626;
                    END_IF;

                    IF TRUE THEN
                        THIS.CallTimers(FALSE);
                        _progress := 427;
                    END_IF;
                END_IF;

                IF _progress = 427 THEN                                                                                     // TemplateTask_20steps_4 running: , <add the detailed description of the current action 8>
                    TaskMessenger.ActivateOnCondition(ULINT#627, _infoTimer.output, eAxoMessageCategory#Warning);
                    IF _infoTimer.output THEN
                        Status.Error.Id := UINT#627;
                    END_IF;

                    IF TRUE THEN
                        THIS.CallTimers(FALSE);
                        _progress := 428;
                    END_IF;
                END_IF;

                IF _progress = 428 THEN                                                                                     // TemplateTask_20steps_4 running: , <add the detailed description of the current action 9>
                    TaskMessenger.ActivateOnCondition(ULINT#628, _infoTimer.output, eAxoMessageCategory#Warning);
                    IF _infoTimer.output THEN
                        Status.Error.Id := UINT#628;
                    END_IF;

                    IF TRUE THEN
                        THIS.CallTimers(FALSE);
                        _progress := 429;
                    END_IF;
                END_IF;

                IF _progress = 429 THEN                                                                                     // TemplateTask_20steps_4 running: , <add the detailed description of the current action 10>
                    TaskMessenger.ActivateOnCondition(ULINT#629, _infoTimer.output, eAxoMessageCategory#Warning);
                    IF _infoTimer.output THEN
                        Status.Error.Id := UINT#629;
                    END_IF;

                    IF TRUE THEN
                        THIS.CallTimers(FALSE);
                        _progress := 430;
                    END_IF;
                END_IF;

                IF _progress = 430 THEN                                                                                     // TemplateTask_20steps_4 running: , <add the detailed description of the current action 11>
                    TaskMessenger.ActivateOnCondition(ULINT#630, _infoTimer.output, eAxoMessageCategory#Warning);
                    IF _infoTimer.output THEN
                        Status.Error.Id := UINT#630;
                    END_IF;

                    IF TRUE THEN
                        THIS.CallTimers(FALSE);
                        _progress := 431;
                    END_IF;
                END_IF;

                IF _progress = 431 THEN                                                                                     // TemplateTask_20steps_4 running: , <add the detailed description of the current action 12>
                    TaskMessenger.ActivateOnCondition(ULINT#631, _infoTimer.output, eAxoMessageCategory#Warning);
                    IF _infoTimer.output THEN
                        Status.Error.Id := UINT#631;
                    END_IF;

                    IF TRUE THEN
                        THIS.CallTimers(FALSE);
                        _progress := 432;
                    END_IF;
                END_IF;

                IF _progress = 432 THEN                                                                                     // TemplateTask_20steps_4 running: , <add the detailed description of the current action 13>
                    TaskMessenger.ActivateOnCondition(ULINT#632, _infoTimer.output, eAxoMessageCategory#Warning);
                    IF _infoTimer.output THEN
                        Status.Error.Id := UINT#632;
                    END_IF;

                    IF TRUE THEN
                        THIS.CallTimers(FALSE);
                        _progress := 433;
                    END_IF;
                END_IF;

                IF _progress = 433 THEN                                                                                     // TemplateTask_20steps_4 running: , <add the detailed description of the current action 14>
                    TaskMessenger.ActivateOnCondition(ULINT#633, _infoTimer.output, eAxoMessageCategory#Warning);
                    IF _infoTimer.output THEN
                        Status.Error.Id := UINT#633;
                    END_IF;

                    IF TRUE THEN
                        THIS.CallTimers(FALSE);
                        _progress := 434;
                    END_IF;
                END_IF;

                IF _progress = 434 THEN                                                                                     // TemplateTask_20steps_4 running: , <add the detailed description of the current action 15>
                    TaskMessenger.ActivateOnCondition(ULINT#634, _infoTimer.output, eAxoMessageCategory#Warning);
                    IF _infoTimer.output THEN
                        Status.Error.Id := UINT#634;
                    END_IF;

                    IF TRUE THEN
                        THIS.CallTimers(FALSE);
                        _progress := 435;
                    END_IF;
                END_IF;

                IF _progress = 435 THEN                                                                                     // TemplateTask_20steps_4 running: , <add the detailed description of the current action 16>
                    TaskMessenger.ActivateOnCondition(ULINT#635, _infoTimer.output, eAxoMessageCategory#Warning);
                    IF _infoTimer.output THEN
                        Status.Error.Id := UINT#635;
                    END_IF;

                    IF TRUE THEN
                        THIS.CallTimers(FALSE);
                        _progress := 436;
                    END_IF;
                END_IF;

                IF _progress = 436 THEN                                                                                     // TemplateTask_20steps_4 running: , <add the detailed description of the current action 17>
                    TaskMessenger.ActivateOnCondition(ULINT#636, _infoTimer.output, eAxoMessageCategory#Warning);
                    IF _infoTimer.output THEN
                        Status.Error.Id := UINT#636;
                    END_IF;

                    IF TRUE THEN
                        THIS.CallTimers(FALSE);
                        _progress := 437;
                    END_IF;
                END_IF;

                IF _progress = 437 THEN                                                                                     // TemplateTask_20steps_4 running: , <add the detailed description of the current action 18>
                    TaskMessenger.ActivateOnCondition(ULINT#637, _infoTimer.output, eAxoMessageCategory#Warning);
                    IF _infoTimer.output THEN
                        Status.Error.Id := UINT#637;
                    END_IF;

                    IF TRUE THEN
                        THIS.CallTimers(FALSE);
                        _progress := 438;
                    END_IF;
                END_IF;

                IF _progress = 438 THEN                                                                                     // TemplateTask_20steps_4 running: , <add the detailed description of the current action 19>
                    TaskMessenger.ActivateOnCondition(ULINT#638, _infoTimer.output, eAxoMessageCategory#Warning);
                    IF _infoTimer.output THEN
                        Status.Error.Id := UINT#638;
                    END_IF;

                    IF TRUE THEN
                        THIS.CallTimers(FALSE);
                        _progress := 439;
                    END_IF;
                END_IF;

                IF _progress = 439 THEN                                                                                     // TemplateTask_20steps_4 running: , <add the detailed description of the current action 20>
                    TemplateTask_20steps_4.DoneWhen(TRUE);
                END_IF;

                THIS.CallTimers(TRUE);

                TemplateTask_20steps_4.ThrowWhen(_errorTimer.output);
                Status.Action.Id := TO_UINT(_progress);
                TemplateTask_20steps_4.ThrowWhen(TemplateTask_20steps_4.Duration >= Config.ErrorTime ,'TemplateTask_20steps_4 error');
            END_IF;
            IF TemplateTask_20steps_4.DoneReached() THEN
                Status.Action.Id :=  UINT#221;
                Status.Error.Id :=  UINT#0;
            ELSIF TemplateTask_20steps_4.ErrorOccured() THEN
                Status.Action.Id :=  UINT#1020;
                Status.Error.Id  :=  UINT#1020;
            ELSIF TemplateTask_20steps_4.AbortTriggered()THEN
                Status.Action.Id :=  UINT#1021;
                Status.Error.Id  :=  UINT#1021;
            END_IF;
            Messenger.ActivateOnCondition(ULINT#1020,TemplateTask_20steps_4.HasError(), eAxoMessageCategory#Error);
            Messenger.ActivateOnCondition(ULINT#1021,TemplateTask_20steps_4.IsAborted(), eAxoMessageCategory#Error);
            Messenger.ActivateOnCondition(ULINT#222,TemplateTask_20steps_4.RestoreTriggered() , eAxoMessageCategory#Error);
            IF TemplateTask_20steps_4.RestoreTriggered() AND _progress >= 420 AND _progress <= 439  THEN
                Status.Action.Id :=  UINT#222;
                _progress := 0;
            END_IF;
            //**************************************************

            //*************TemplateTask_20steps_5***************
            TemplateTask_20steps_5.SetIsDisabled(FALSE);
            IF TemplateTask_20steps_5.StartTriggered() THEN
                Status.Action.Id :=  UINT#240;
            END_IF;
            Messenger.ActivateOnCondition(ULINT#240,TemplateTask_20steps_5.IsBusy(), eAxoMessageCategory#Info);
            Messenger.ActivateOnCondition(ULINT#241,TemplateTask_20steps_5.IsDone(), eAxoMessageCategory#Info);
            IF TemplateTask_20steps_5.Execute(THIS) THEN
                IF _progress = 0 THEN
                    Status.Error.Id := UINT#0;
                    TaskMessenger.Restore();
                    THIS.CallTimers(FALSE);
                    _progress := 440;
                END_IF;

                IF _progress = 440 THEN                                                                                     // TemplateTask_20steps_5 running: , <add the detailed description of the current action 1>
                    TaskMessenger.ActivateOnCondition(ULINT#640, _infoTimer.output, eAxoMessageCategory#Warning);
                    IF _infoTimer.output THEN
                        Status.Error.Id := UINT#640;
                    END_IF;

                    IF TRUE THEN
                        THIS.CallTimers(FALSE);
                        _progress := 441;
                    END_IF;
                END_IF;

                IF _progress = 441 THEN                                                                                     // TemplateTask_20steps_5 running , <add the detailed description of the current action 2>
                    TaskMessenger.ActivateOnCondition(ULINT#641, _infoTimer.output, eAxoMessageCategory#Warning);
                    IF _infoTimer.output THEN
                        Status.Error.Id := UINT#641;
                    END_IF;

                    IF TRUE THEN
                        THIS.CallTimers(FALSE);
                        _progress := 442;
                    END_IF;
                END_IF;

                IF _progress = 442 THEN                                                                                     // TemplateTask_20steps_5 running: , <add the detailed description of the current action 3>
                    TaskMessenger.ActivateOnCondition(ULINT#642, _infoTimer.output, eAxoMessageCategory#Warning);
                    IF _infoTimer.output THEN
                        Status.Error.Id := UINT#642;
                    END_IF;

                    IF TRUE THEN
                        THIS.CallTimers(FALSE);
                        _progress := 443;
                    END_IF;
                END_IF;

                IF _progress = 443 THEN                                                                                     // TemplateTask_20steps_5 running: , <add the detailed description of the current action 4>
                    TaskMessenger.ActivateOnCondition(ULINT#643, _infoTimer.output, eAxoMessageCategory#Warning);
                    IF _infoTimer.output THEN
                        Status.Error.Id := UINT#643;
                    END_IF;

                    IF TRUE THEN
                        THIS.CallTimers(FALSE);
                        _progress := 444;
                    END_IF;
                END_IF;

                IF _progress = 444 THEN                                                                                     // TemplateTask_20steps_5 running: , <add the detailed description of the current action 5>
                    TaskMessenger.ActivateOnCondition(ULINT#644, _infoTimer.output, eAxoMessageCategory#Warning);
                    IF _infoTimer.output THEN
                        Status.Error.Id := UINT#644;
                    END_IF;

                    IF TRUE THEN
                        THIS.CallTimers(FALSE);
                        _progress := 445;
                    END_IF;
                END_IF;

                IF _progress = 445 THEN                                                                                     // TemplateTask_20steps_5 running: , <add the detailed description of the current action 6>
                    TaskMessenger.ActivateOnCondition(ULINT#645, _infoTimer.output, eAxoMessageCategory#Warning);
                    IF _infoTimer.output THEN
                        Status.Error.Id := UINT#645;
                    END_IF;

                    IF TRUE THEN
                        THIS.CallTimers(FALSE);
                        _progress := 446;
                    END_IF;
                END_IF;

                IF _progress = 446 THEN                                                                                     // TemplateTask_20steps_5 running: , <add the detailed description of the current action 7>
                    TaskMessenger.ActivateOnCondition(ULINT#646, _infoTimer.output, eAxoMessageCategory#Warning);
                    IF _infoTimer.output THEN
                        Status.Error.Id := UINT#646;
                    END_IF;

                    IF TRUE THEN
                        THIS.CallTimers(FALSE);
                        _progress := 447;
                    END_IF;
                END_IF;

                IF _progress = 447 THEN                                                                                     // TemplateTask_20steps_5 running: , <add the detailed description of the current action 8>
                    TaskMessenger.ActivateOnCondition(ULINT#647, _infoTimer.output, eAxoMessageCategory#Warning);
                    IF _infoTimer.output THEN
                        Status.Error.Id := UINT#647;
                    END_IF;

                    IF TRUE THEN
                        THIS.CallTimers(FALSE);
                        _progress := 448;
                    END_IF;
                END_IF;

                IF _progress = 448 THEN                                                                                     // TemplateTask_20steps_5 running: , <add the detailed description of the current action 9>
                    TaskMessenger.ActivateOnCondition(ULINT#648, _infoTimer.output, eAxoMessageCategory#Warning);
                    IF _infoTimer.output THEN
                        Status.Error.Id := UINT#648;
                    END_IF;

                    IF TRUE THEN
                        THIS.CallTimers(FALSE);
                        _progress := 449;
                    END_IF;
                END_IF;

                IF _progress = 449 THEN                                                                                     // TemplateTask_20steps_5 running: , <add the detailed description of the current action 10>
                    TaskMessenger.ActivateOnCondition(ULINT#649, _infoTimer.output, eAxoMessageCategory#Warning);
                    IF _infoTimer.output THEN
                        Status.Error.Id := UINT#649;
                    END_IF;

                    IF TRUE THEN
                        THIS.CallTimers(FALSE);
                        _progress := 450;
                    END_IF;
                END_IF;

                IF _progress = 450 THEN                                                                                     // TemplateTask_20steps_5 running: , <add the detailed description of the current action 11>
                    TaskMessenger.ActivateOnCondition(ULINT#650, _infoTimer.output, eAxoMessageCategory#Warning);
                    IF _infoTimer.output THEN
                        Status.Error.Id := UINT#650;
                    END_IF;

                    IF TRUE THEN
                        THIS.CallTimers(FALSE);
                        _progress := 451;
                    END_IF;
                END_IF;

                IF _progress = 451 THEN                                                                                     // TemplateTask_20steps_5 running: , <add the detailed description of the current action 12>
                    TaskMessenger.ActivateOnCondition(ULINT#651, _infoTimer.output, eAxoMessageCategory#Warning);
                    IF _infoTimer.output THEN
                        Status.Error.Id := UINT#651;
                    END_IF;

                    IF TRUE THEN
                        THIS.CallTimers(FALSE);
                        _progress := 452;
                    END_IF;
                END_IF;

                IF _progress = 452 THEN                                                                                     // TemplateTask_20steps_5 running: , <add the detailed description of the current action 13>
                    TaskMessenger.ActivateOnCondition(ULINT#652, _infoTimer.output, eAxoMessageCategory#Warning);
                    IF _infoTimer.output THEN
                        Status.Error.Id := UINT#652;
                    END_IF;

                    IF TRUE THEN
                        THIS.CallTimers(FALSE);
                        _progress := 453;
                    END_IF;
                END_IF;

                IF _progress = 453 THEN                                                                                     // TemplateTask_20steps_5 running: , <add the detailed description of the current action 14>
                    TaskMessenger.ActivateOnCondition(ULINT#653, _infoTimer.output, eAxoMessageCategory#Warning);
                    IF _infoTimer.output THEN
                        Status.Error.Id := UINT#653;
                    END_IF;

                    IF TRUE THEN
                        THIS.CallTimers(FALSE);
                        _progress := 454;
                    END_IF;
                END_IF;

                IF _progress = 454 THEN                                                                                     // TemplateTask_20steps_5 running: , <add the detailed description of the current action 15>
                    TaskMessenger.ActivateOnCondition(ULINT#654, _infoTimer.output, eAxoMessageCategory#Warning);
                    IF _infoTimer.output THEN
                        Status.Error.Id := UINT#654;
                    END_IF;

                    IF TRUE THEN
                        THIS.CallTimers(FALSE);
                        _progress := 455;
                    END_IF;
                END_IF;

                IF _progress = 455 THEN                                                                                     // TemplateTask_20steps_5 running: , <add the detailed description of the current action 16>
                    TaskMessenger.ActivateOnCondition(ULINT#655, _infoTimer.output, eAxoMessageCategory#Warning);
                    IF _infoTimer.output THEN
                        Status.Error.Id := UINT#655;
                    END_IF;

                    IF TRUE THEN
                        THIS.CallTimers(FALSE);
                        _progress := 456;
                    END_IF;
                END_IF;

                IF _progress = 456 THEN                                                                                     // TemplateTask_20steps_5 running: , <add the detailed description of the current action 17>
                    TaskMessenger.ActivateOnCondition(ULINT#656, _infoTimer.output, eAxoMessageCategory#Warning);
                    IF _infoTimer.output THEN
                        Status.Error.Id := UINT#656;
                    END_IF;

                    IF TRUE THEN
                        THIS.CallTimers(FALSE);
                        _progress := 457;
                    END_IF;
                END_IF;

                IF _progress = 457 THEN                                                                                     // TemplateTask_20steps_5 running: , <add the detailed description of the current action 18>
                    TaskMessenger.ActivateOnCondition(ULINT#657, _infoTimer.output, eAxoMessageCategory#Warning);
                    IF _infoTimer.output THEN
                        Status.Error.Id := UINT#657;
                    END_IF;

                    IF TRUE THEN
                        THIS.CallTimers(FALSE);
                        _progress := 458;
                    END_IF;
                END_IF;

                IF _progress = 458 THEN                                                                                     // TemplateTask_20steps_5 running: , <add the detailed description of the current action 19>
                    TaskMessenger.ActivateOnCondition(ULINT#658, _infoTimer.output, eAxoMessageCategory#Warning);
                    IF _infoTimer.output THEN
                        Status.Error.Id := UINT#658;
                    END_IF;

                    IF TRUE THEN
                        THIS.CallTimers(FALSE);
                        _progress := 459;
                    END_IF;
                END_IF;

                IF _progress = 459 THEN                                                                                     // TemplateTask_20steps_5 running: , <add the detailed description of the current action 20>
                    TemplateTask_20steps_5.DoneWhen(TRUE);
                END_IF;

                THIS.CallTimers(TRUE);

                TemplateTask_20steps_5.ThrowWhen(_errorTimer.output);
                Status.Action.Id := TO_UINT(_progress);
                TemplateTask_20steps_5.ThrowWhen(TemplateTask_20steps_5.Duration >= Config.ErrorTime ,'TemplateTask_20steps_5 error.');
            END_IF;
            IF TemplateTask_20steps_5.DoneReached() THEN
                Status.Action.Id :=  UINT#241;
                Status.Error.Id :=  UINT#0;
            ELSIF TemplateTask_20steps_5.ErrorOccured() THEN
                Status.Action.Id :=  UINT#1040;
                Status.Error.Id  :=  UINT#1040;
            ELSIF TemplateTask_20steps_5.AbortTriggered()THEN
                Status.Action.Id :=  UINT#1041;
                Status.Error.Id  :=  UINT#1041;
            END_IF;
            Messenger.ActivateOnCondition(ULINT#1040,TemplateTask_20steps_5.HasError(), eAxoMessageCategory#Error);
            Messenger.ActivateOnCondition(ULINT#1041,TemplateTask_20steps_5.IsAborted(), eAxoMessageCategory#Error);
            Messenger.ActivateOnCondition(ULINT#242,TemplateTask_20steps_5.RestoreTriggered() , eAxoMessageCategory#Error);
            IF TemplateTask_20steps_5.RestoreTriggered() AND _progress >= 440 AND _progress <= 459  THEN
                Status.Action.Id :=  UINT#242;
                _progress := 0;
            END_IF;
            //**************************************************

            //*************TemplateTask_20steps_6***************
            TemplateTask_20steps_6.SetIsDisabled(FALSE);
            IF TemplateTask_20steps_6.StartTriggered() THEN
                Status.Action.Id :=  UINT#260;
            END_IF;
            Messenger.ActivateOnCondition(ULINT#260,TemplateTask_20steps_6.IsBusy(), eAxoMessageCategory#Info);
            Messenger.ActivateOnCondition(ULINT#261,TemplateTask_20steps_6.IsDone(), eAxoMessageCategory#Info);
            IF TemplateTask_20steps_6.Execute(THIS) THEN
                IF _progress = 0 THEN
                    Status.Error.Id := UINT#0;
                    TaskMessenger.Restore();
                    THIS.CallTimers(FALSE);
                    _progress := 460;
                END_IF;

                IF _progress = 460 THEN                                                                                     // TemplateTask_20steps_6 running: , <add the detailed description of the current action 1>
                    TaskMessenger.ActivateOnCondition(ULINT#660, _infoTimer.output, eAxoMessageCategory#Warning);
                    IF _infoTimer.output THEN
                        Status.Error.Id := UINT#660;
                    END_IF;

                    IF TRUE THEN
                        THIS.CallTimers(FALSE);
                        _progress := 461;
                    END_IF;
                END_IF;

                IF _progress = 461 THEN                                                                                     // TemplateTask_20steps_6 running: , <add the detailed description of the current action 2>
                    TaskMessenger.ActivateOnCondition(ULINT#661, _infoTimer.output, eAxoMessageCategory#Warning);
                    IF _infoTimer.output THEN
                        Status.Error.Id := UINT#661;
                    END_IF;

                    IF TRUE THEN
                        THIS.CallTimers(FALSE);
                        _progress := 462;
                    END_IF;
                END_IF;

                IF _progress = 462 THEN                                                                                     // TemplateTask_20steps_6 running: , <add the detailed description of the current action 3>
                    TaskMessenger.ActivateOnCondition(ULINT#662, _infoTimer.output, eAxoMessageCategory#Warning);
                    IF _infoTimer.output THEN
                        Status.Error.Id := UINT#662;
                    END_IF;

                    IF TRUE THEN
                        THIS.CallTimers(FALSE);
                        _progress := 463;
                    END_IF;
                END_IF;

                IF _progress = 463 THEN                                                                                     // TemplateTask_20steps_6 running: , <add the detailed description of the current action 4>
                    TaskMessenger.ActivateOnCondition(ULINT#663, _infoTimer.output, eAxoMessageCategory#Warning);
                    IF _infoTimer.output THEN
                        Status.Error.Id := UINT#663;
                    END_IF;

                    IF TRUE THEN
                        THIS.CallTimers(FALSE);
                        _progress := 464;
                    END_IF;
                END_IF;

                IF _progress = 464 THEN                                                                                     // TemplateTask_20steps_6 running: , <add the detailed description of the current action 5>
                    TaskMessenger.ActivateOnCondition(ULINT#664, _infoTimer.output, eAxoMessageCategory#Warning);
                    IF _infoTimer.output THEN
                        Status.Error.Id := UINT#664;
                    END_IF;

                    IF TRUE THEN
                        THIS.CallTimers(FALSE);
                        _progress := 465;
                    END_IF;
                END_IF;

                IF _progress = 465 THEN                                                                                     // TemplateTask_20steps_6 running: , <add the detailed description of the current action 6>
                    TaskMessenger.ActivateOnCondition(ULINT#665, _infoTimer.output, eAxoMessageCategory#Warning);
                    IF _infoTimer.output THEN
                        Status.Error.Id := UINT#665;
                    END_IF;

                    IF TRUE THEN
                        THIS.CallTimers(FALSE);
                        _progress := 466;
                    END_IF;
                END_IF;

                IF _progress = 466 THEN                                                                                     // TemplateTask_20steps_6 running: , <add the detailed description of the current action 7>
                    TaskMessenger.ActivateOnCondition(ULINT#666, _infoTimer.output, eAxoMessageCategory#Warning);
                    IF _infoTimer.output THEN
                        Status.Error.Id := UINT#666;
                    END_IF;

                    IF TRUE THEN
                        THIS.CallTimers(FALSE);
                        _progress := 467;
                    END_IF;
                END_IF;

                IF _progress = 467 THEN                                                                                     // TemplateTask_20steps_6 running: , <add the detailed description of the current action 8>
                    TaskMessenger.ActivateOnCondition(ULINT#667, _infoTimer.output, eAxoMessageCategory#Warning);
                    IF _infoTimer.output THEN
                        Status.Error.Id := UINT#667;
                    END_IF;

                    IF TRUE THEN
                        THIS.CallTimers(FALSE);
                        _progress := 468;
                    END_IF;
                END_IF;

                IF _progress = 468 THEN                                                                                     // TemplateTask_20steps_6 running: , <add the detailed description of the current action 9>
                    TaskMessenger.ActivateOnCondition(ULINT#668, _infoTimer.output, eAxoMessageCategory#Warning);
                    IF _infoTimer.output THEN
                        Status.Error.Id := UINT#668;
                    END_IF;

                    IF TRUE THEN
                        THIS.CallTimers(FALSE);
                        _progress := 469;
                    END_IF;
                END_IF;

                IF _progress = 469 THEN                                                                                     // TemplateTask_20steps_6 running: , <add the detailed description of the current action 10>
                    TaskMessenger.ActivateOnCondition(ULINT#669, _infoTimer.output, eAxoMessageCategory#Warning);
                    IF _infoTimer.output THEN
                        Status.Error.Id := UINT#669;
                    END_IF;

                    IF TRUE THEN
                        THIS.CallTimers(FALSE);
                        _progress := 470;
                    END_IF;
                END_IF;

                IF _progress = 470 THEN                                                                                     // TemplateTask_20steps_6 running: , <add the detailed description of the current action 11>
                    TaskMessenger.ActivateOnCondition(ULINT#670, _infoTimer.output, eAxoMessageCategory#Warning);
                    IF _infoTimer.output THEN
                        Status.Error.Id := UINT#670;
                    END_IF;

                    IF TRUE THEN
                        THIS.CallTimers(FALSE);
                        _progress := 471;
                    END_IF;
                END_IF;

                IF _progress = 471 THEN                                                                                     // TemplateTask_20steps_6 running: , <add the detailed description of the current action 12>
                    TaskMessenger.ActivateOnCondition(ULINT#671, _infoTimer.output, eAxoMessageCategory#Warning);
                    IF _infoTimer.output THEN
                        Status.Error.Id := UINT#671;
                    END_IF;

                    IF TRUE THEN
                        THIS.CallTimers(FALSE);
                        _progress := 472;
                    END_IF;
                END_IF;

                IF _progress = 472 THEN                                                                                     // TemplateTask_20steps_6 running: , <add the detailed description of the current action 13>
                    TaskMessenger.ActivateOnCondition(ULINT#672, _infoTimer.output, eAxoMessageCategory#Warning);
                    IF _infoTimer.output THEN
                        Status.Error.Id := UINT#672;
                    END_IF;

                    IF TRUE THEN
                        THIS.CallTimers(FALSE);
                        _progress := 473;
                    END_IF;
                END_IF;

                IF _progress = 473 THEN                                                                                     // TemplateTask_20steps_6 running: , <add the detailed description of the current action 14>
                    TaskMessenger.ActivateOnCondition(ULINT#673, _infoTimer.output, eAxoMessageCategory#Warning);
                    IF _infoTimer.output THEN
                        Status.Error.Id := UINT#673;
                    END_IF;

                    IF TRUE THEN
                        THIS.CallTimers(FALSE);
                        _progress := 474;
                    END_IF;
                END_IF;

                IF _progress = 474 THEN                                                                                     // TemplateTask_20steps_6 running: , <add the detailed description of the current action 15>
                    TaskMessenger.ActivateOnCondition(ULINT#674, _infoTimer.output, eAxoMessageCategory#Warning);
                    IF _infoTimer.output THEN
                        Status.Error.Id := UINT#674;
                    END_IF;

                    IF TRUE THEN
                        THIS.CallTimers(FALSE);
                        _progress := 475;
                    END_IF;
                END_IF;
